FUNCTION_BLOCK FB_CANMessageHandler
VAR_INPUT
	Outputs 	: REFERENCE TO CANTXQUEUESTRUCT_N_1; // CAN muuttujat
	Inputs 		: REFERENCE TO CANRXQUEUESTRUCT_N_1;
	
	fVoltage_A	: REAL; // Jännite A realina
	fVoltage_B	: REAL; // Jännite B realina
END_VAR
VAR
	i				: DINT;
	MessageReceived : CANQUEUE;
	MessageToSend	: CANQUEUE;
	NumberOfMessagesToSend	: UINT := 1;
	wV_a,wV_b		: WORD;
END_VAR


wV_a := F_VoltageToWord(Voltage_In := fVoltage_A);
wV_b := F_VoltageToWord(Voltage_In := fVoltage_B);

MessageToSend := F_GenerateCANMessage(cobID := 4, V_a := wV_a, V_b := wV_b);

IF Outputs.TxCounter = Inputs.TxCounter THEN
   	Outputs.TxMessages[0] := MessageToSend;
    Outputs.NoOfTxMessages := NumberOfMessagesToSend;
    Outputs.TxCounter := Outputs.TxCounter + 1;
END_IF

END_FUNCTION_BLOCK

(* stored: Version 1.1.0.1, ProductVersion 3.1.4022.17
   POU FB_CANMessageHandler: Id {ad659beb-b876-4d1c-acaf-e86a9ddd6681}, SpecialFunc None *)
